{attribute 'GeneratedUsingTerminal: EPP2339-0021-0016'}
{attribute addProperty BoxType "EPP2339-0021-0016"}
{attribute addProperty Id "InputAT %I*BOOL1"}
{attribute addProperty CRC "2198356929"}
{attribute addProperty Size "1"}
TYPE Channel_830843C1 EXTENDS InputBase_8311D824 :
STRUCT
	{attribute addProperty Name "Input"}
	Input AT %I* : BOOL;
END_STRUCT
END_TYPE

(* stored: Version 1.2.0.0, ProductVersion 3.1.4024.9
   DUT Channel_830843C1: Id {a9bcb12c-8800-4ee6-9f50-69409b85273a} *)
